// TIA Portal V20 export
DATA_BLOCK "CallEquipment_DB"   // DB90
{ DB_Accessible_From_OPC_UA := 'FALSE' }
// stored: AssignedProDiagFB Unit1.Em9.ProDiag, DBAccessibleFromOPCUA false, DBAccessibleFromWebserver false, InstanceOfName Unit1.Em9.CallEquipment, InstanceOfType FB, Namespace Unit1.Em9
"Unit1.Em9.CallEquipment"
   // VAR_INPUT
   //    ZoneOperationEnable { ExternalWritable := 'False'} : "LWONIK_typeSafetyZoneManualOperation";
   // END_VAR
   // VAR_IN_OUT
   //    unitStatus : "LAF_typeUnitStatus";
   //    emFeedback : "LUC_typeEmFeedback";
   //    unitAlarmDB : "LAF_typeAlarms";
   // END_VAR
   // VAR
   //    InstSequenceVision { ExternalWritable := 'False'} : "Unit1.Em9.Sequence_1_Vision";
   //    instVisionHomeJob1 { ExternalWritable := 'False'} : "LAF_SelectJob";
   //    instVisionLoadJob2 { ExternalWritable := 'False'} : "LAF_SelectJob";
   //    instVisionInspectionJob3 { ExternalWritable := 'False'} : "LAF_SelectJob";
   //    instVisionUnloadJob4 { ExternalWritable := 'False'} : "LAF_SelectJob";
   //    instGRnR_visionLoadJob2 { ExternalWritable := 'False'; S7_SetPoint := 'True'} : "LAF_SelectJob";
   //    instGRnR_visionInspectionJob3 { ExternalWritable := 'False'; S7_SetPoint := 'True'} : "LAF_SelectJob";
   //    instGRnR_visionUnloadJob4 { ExternalWritable := 'False'; S7_SetPoint := 'True'} : "LAF_SelectJob";
   //    instCmVisionJRDetect { ExternalWritable := 'False'} : "LBC_DigitalSignalCn";
   //    instCmVisionStageLiftUpDown { ExternalWritable := 'False'} : "LBC_TwoWayActuatorCn";
   //    instCmVisionLightUpDown { ExternalWritable := 'False'} : "LBC_TwoWayActuatorCn";
   //    instVisionConversion { ExternalWritable := 'False'} : "LER_Vision_XGX2000_Conversion";
   //    instVisionHistory { ExternalWritable := 'False'} : "LER_visionHistory";
   //    instVisionHistoryRnR { ExternalWritable := 'False'} : "LER_visionHistory";
   //    instManageAlarms { ExternalWritable := 'False'} : "LAF_ManageAlarms";
   //    instEventsPFE { ExternalWritable := 'False'} : "Unit1.Em9.EventsPFE";
   //    statUnitStatus { ExternalWritable := 'False'} : "LAF_typeUnitStatus";
   //    statPartData { ExternalWritable := 'False'} : "LER_typePartData";
   //    statDataDelete { ExternalWritable := 'False'} : "LER_typePartData";
   //    statHistoryDeleteData { ExternalWritable := 'False'} : "LER_typeVisionHistory";
   //    statTonTime { ExternalWritable := 'False'} : Array[0..999] of TON_TIME;
   //    statTofTime { ExternalWritable := 'False'} : Array[0..9] of TOF_TIME;
   //    statPulse { ExternalWritable := 'False'} : Array[0..999] of Bool;
   //    statVision_GaugeRnR : Struct
   //       currentCount : Int;
   //       processCount : Int := 50;
   //       Ongoing : Bool;
   //       Complete : Bool;
   //    END_STRUCT;
   //    statTraceCode { ExternalWritable := 'False'} : String[18];
   //    statEnableManualCmds { ExternalWritable := 'False'} : Bool;
   //    statNomalMode { ExternalWritable := 'False'} : Bool;
   //    statCodeGenerate { ExternalWritable := 'False'} : Bool;
   //    statGaugeRnRComplete { ExternalWritable := 'False'} : Bool;
   //    "*** Interlock TwoWay ***" { S7_SetPoint := 'True'} : "LER_Axis_Homing";
   //    instCmVisionStageLiftUpDownInterlock { S7_SetPoint := 'True'} : Array[0..2] of "LER_Actuator";
   //    instCmVisionLightUpDownInterlock { S7_SetPoint := 'True'} : Array[0..2] of "LER_Actuator";
   //    VisionStageLiftUpDown_Inpos : Array[0..2] of Struct
   //       "Int" : Array[1..10] of Bool;
   //    END_STRUCT;
   //    VisionLightUpDown_Inpos : Array[0..2] of Struct
   //       "Int" : Array[1..10] of Bool;
   //    END_STRUCT;
   //    instVisionControl { S7_SetPoint := 'True'} : "LER_Vision_XGX2000";
   //    Sequence_10_GaugeRnRVision_Instance { S7_SetPoint := 'True'} : "Unit1.Em9.Sequence_10_GaugeRnRVision";
   //    citi_Ptrig : Array[0..20] of Bool;
   //    citiTon : Array[0..20] of TON_TIME;
   //    citi : Time;
   //    citiTest : Array[0..20] of Bool;
   // END_VAR
BEGIN
END_DATA_BLOCK
